// TwinCAT 3 PLC project ProjectPLC
// ProgramVersion: 3.1.4020.2
// libraries:
//   Tc2_Standard, * (Beckhoff Automation GmbH)
//   Tc2_System, * (Beckhoff Automation GmbH)
//   Tc3_Module, * (Beckhoff Automation GmbH)
//   VisuDialogs, * (System)
// project tree:
//   / GlobalTextList.TcGTLO, PlcTask.TcTTO, Visualization Manager.TcVMO (not stored), VISU_TASK.TcTTO
//   POUs/ MAIN.TcPOU
//   VISUs/ Visualization.TcVIS
// real-time tasks:
//   TASK PlcTask: cycle T#10ms, priority 20, ADS port 350
//   TASK VISU_TASK: cycle T#200000us, priority 30, ADS port 351
// I/O:
//   DEVICE Device 1 (EtherCAT) (disabled), AmsNetId 5.42.99.255.2.1
//     Term 1 (EK1200) [EK1200-5000 EtherCAT Power supply (2A E-Bus)]
//       Term 2 (EL2008) [EL2008 8Ch. Dig. Output 24V, 0.5A]
//       Term 3 (EL3044) [EL3044 4Ch. Ana. Input 0-20mA]
//       Term 4 (EL3044) [EL3044 4Ch. Ana. Input 0-20mA]
//       Term 5 (EL3044) [EL3044 4Ch. Ana. Input 0-20mA]
//       Term 6 (EL1004) [EL1004 4Ch. Dig. Input 24V, 3ms]
//       Term 7 (EL1004) [EL1004 4Ch. Dig. Input 24V, 3ms]

CONFIGURATION ProjectPLC
    RESOURCE PLC ON TwinCAT3
        TASK PlcTask(INTERVAL := T#10ms, PRIORITY := 20);
        TASK VISU_TASK(INTERVAL := T#200000us, PRIORITY := 30);
        PROGRAM MAIN WITH PlcTask : MAIN;
        PROGRAM VisuElems_Visu_Prg WITH VISU_TASK : VisuElems.Visu_Prg;
    END_RESOURCE
END_CONFIGURATION

// ---- POUs/MAIN.TcPOU
PROGRAM MAIN
VAR
	udiDeviceID 			: UDINT 	:= 1;
	sTargetNetID 			: STRING 	:= '192.168.1.20.1.1';
	sSlaveDescriptionPath	: STRING 	:= 'C:\TwinCAT\3.1\Config\Io\EtherCAT';
	udiZoomFactor 			: UDINT 	:= 3;
	bReadOnly 				: BOOL;
	bSowSlaveInfo			: BOOL;
	bShowOnlineTopology		: BOOL;
	bRefresh 				: BOOL;
	
END_VAR

;

END_PROGRAM

// ---- GlobalTextList.TcGTLO
TEXTLIST GlobalTextList
  5 = '%d'
  3 = '%s'
  6 = 'Device ID'
  7 = 'EtherCAT Desc'
  8 = 'Read Only'
  1 = 'Refresh'
  0 = 'Show Online Topology'
  9 = 'Show Slave Info'
  2 = 'Target Net ID'
  4 = 'Zoom Factor'
END_TEXTLIST

// ---- VISUs/Visualization.TcVIS
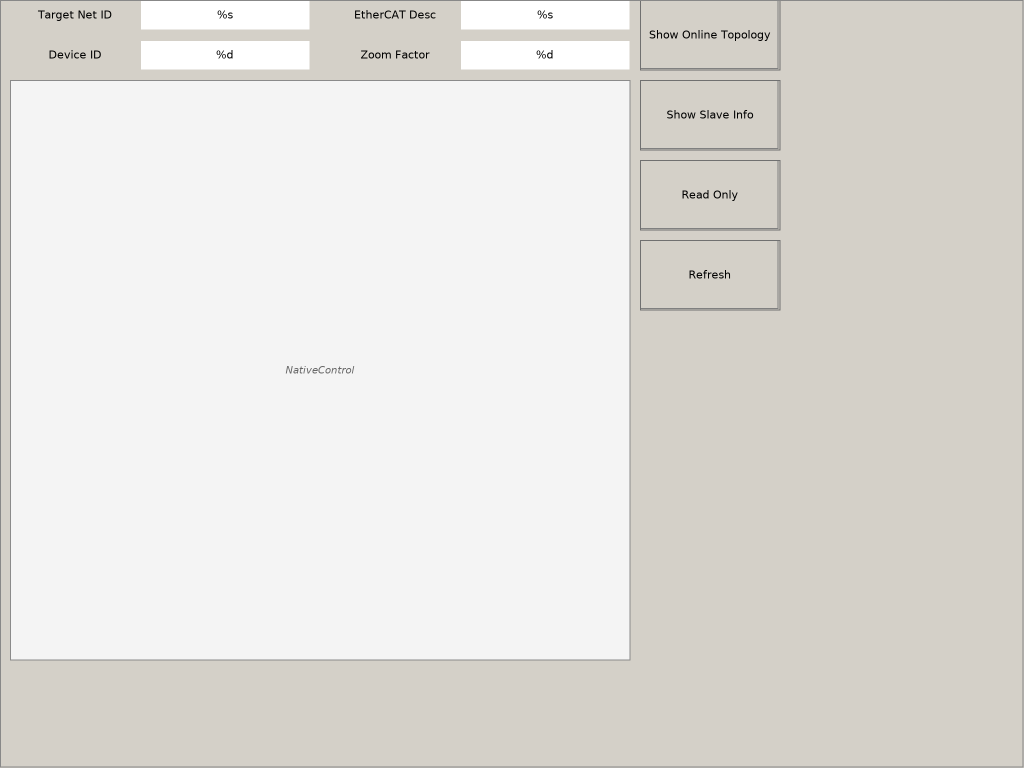
VISUALIZATION Visualization  // 1024x768
    NativeControl (10,80 620x580)
        Calls[0]: Method=TargetNetId, Method=ShowOnlineTopology, Variable=MAIN.bShowOnlineTopology
        Parameters[0]: Var=MAIN.sTargetNetID, Var=MAIN.udiDeviceID, Var=MAIN.udiZoomFactor, Var=MAIN.bSowSlaveInfo, Var=MAIN.sSlaveDescriptionPath, Var=MAIN.bReadOnly
        Calls[1]: Method=DeviceId, Method=ZoomFactor, Variable=MAIN.bRefresh
        Calls[2]: Method=SlaveDescriptionPath, Method=ShowSlaveInfo, Variable=MAIN.bSowSlaveInfo
        Calls[3]: Method=ReadOnly, Variable=MAIN.bRefresh
        p3873840581: EcTopology.EcTopologyCtrl.1
    Button (640,0 140x70), "Show Online Topology"
        tap MAIN.bShowOnlineTopology
    Textfield (140,0 170x30), "%s", text variable: MAIN.sTargetNetID
        OnMouseClick: write the text variable via Default
    Label (0,0 150x30), "Target Net ID"
    Textfield (140,40 170x30), "%d", text variable: MAIN.udiDeviceID
        OnMouseClick: write the text variable via Default
    Label (0,40 150x30), "Device ID"
    Textfield (460,0 170x30), "%s", text variable: MAIN.sSlaveDescriptionPath
        OnMouseClick: write the text variable via Default
    Label (320,0 150x30), "EtherCAT Desc"
    Textfield (460,40 170x30), "%d", text variable: MAIN.udiZoomFactor
        OnMouseClick: write the text variable via Default
    Label (320,40 150x30), "Zoom Factor"
    Button (640,80 140x70), "Show Slave Info"
        toggle MAIN.bSowSlaveInfo
    Button (640,160 140x70), "Read Only"
        tap MAIN.bRefresh
    Button (640,240 140x70), "Refresh"
        tap MAIN.bRefresh
END_VISUALIZATION
